Fanuc KAREL source: ka00131.KL

-- PROVISIONAL review KL for V940-1; original PC SHA256 b8f9c8717b259d3691502ae958b8e214ee0c3d72e437eb694b7a45b570e7573f
-- Incomplete behavior may be omitted. Consult companion uncertainty JSON. Do not deploy.
PROGRAM KA00131
%NOLOCKGROUP
-- UNRESOLVED_DECL SRC type=002018
-- UNRESOLVED_DECL DST type=002018
BEGIN
  -- V9_ZERO_TABLE_METADATA_HINT layout=0001; no indexed target words; source/name/runtime held
  -- UNRESOLVED_PC offsets 5-19; opcodes 2E,22,9D,33,B2
  -- UNRESOLVED_PC offsets 24-42; opcodes 22,9D,33,B1,22,9D,33,B2
  -- UNRESOLVED_PC offsets 47-51; opcodes 7F
END KA00131
